FUNCTION_BLOCK FB_MQTT
VAR_INPUT
END_VAR
VAR_OUTPUT
END_VAR
VAR
END_VAR

END_FUNCTION_BLOCK

(* stored: Version 1.1.0.1, ProductVersion 3.1.4024.9
   POU FB_MQTT: Id {81d5f795-0385-40e6-8396-c56834c61a6c}, SpecialFunc None *)
